Staubli VAL3: GetToolParam6x.pgx

program GetToolParam6x(num& arrayValue[])
begin
  //*******************************************************************************
  //*   ______
  //*  / _____) /|
  //* | |      / /
  //* | | /\  / /
  //* | | \ \/ /  _      Copyright (c) KEOLABS, 2016
  //* | |  \__/  | |        http://www.keolabs.com
  //* | |________| |
  //*  \__________/
  //*
  //********************************************************************************
  //*@file          : GetToolParam6x
  //*@author        : Yves Ragot
  //*@version       : $Id: GetToolParam6x.pgx 1490 2016-12-14 15:39:12Z yves $
  //*@brief         : Get the current tool parameters
  //*
  //*******************************************************************************/

 // get Cartesian parameters and converts to 1/10 mm
  arrayValue[0] = tCurrentTool.trsf.x * 10
  arrayValue[1] = tCurrentTool.trsf.y * 10
  arrayValue[2] = tCurrentTool.trsf.z * 10
  arrayValue[3] = tCurrentTool.trsf.rx * 10
  arrayValue[4] = tCurrentTool.trsf.ry * 10
  arrayValue[5] = tCurrentTool.trsf.rz * 10

end
